(* PLC project conveyor, truST trust-runtime 0.24.54 *)
(* stored: creationDateTime 1786456263Z *)

TYPE XY : STRUCT
  X : lreal;
  Y : lreal;
END_STRUCT;
END_TYPE

FUNCTION RotateSquarePoints : XYPoints
VAR_IN_OUT
    Square : XYPoints;
END_VAR
VAR
   X : LREAL;
   Y : LREAL;
   I : INT;
END_VAR
FOR I := 0 TO 3 DO 
    X := Square[I].X;
    Y := Square[I].Y;
    Square[I] := RotateXY(
    X := X,
    Y := Y,
    THETA := 90.0
    );
END_FOR
RotateSquarePoints := Square;
END_FUNCTION

FUNCTION RotateSquarePoints : XYPoints
VAR_IN_OUT
    Square : XYPoints;
END_VAR
VAR
   X : LREAL;
   Y : LREAL;
   I : INT;
END_VAR
FOR I := 0 TO 3 DO 
    X := Square[I].X;
    Y := Square[I].Y;
    Square[I] := RotateXY(
    X := X,
    Y := Y,
    THETA := 90.0
    );
END_FOR
RotateSquarePoints := Square;
END_FUNCTION
END_FUNCTION

FUNCTION RotateXY : XY
VAR_INPUT
    X : LREAL;
    Y : LREAL;
    THETA : LREAL;
END_VAR
VAR
    Out : XY;
    SinM : LREAL;
    CosM : LREAL;
    THETA_RAD : LREAL;
END_VAR 
   
   THETA_RAD := REAL_TO_LREAL(
    RAD(
        LREAL_TO_REAL(THETA)
        )
    );  
   SinM := SIN(THETA_RAD);
   Cosm := COS(THETA_RAD);
   Out.X := X * CosM - Y * SinM;
   Out.Y := X * SinM + Y * CosM;
   RotateXY := Out;
END_FUNCTION

FUNCTION RotateXY : XY
VAR_INPUT
    X : LREAL;
    Y : LREAL;
    THETA : LREAL;
END_VAR
VAR
    Out : XY;
    SinM : LREAL;
    CosM : LREAL;
    THETA_RAD : LREAL;
END_VAR 
   
   THETA_RAD := REAL_TO_LREAL(
    RAD(
        LREAL_TO_REAL(THETA)
        )
    );  
   SinM := SIN(THETA_RAD);
   Cosm := COS(THETA_RAD);
   Out.X := X * CosM - Y * SinM;
   Out.Y := X * SinM + Y * CosM;
   RotateXY := Out;
END_FUNCTION
END_FUNCTION

FUNCTION SquarePoints : XYPoints
VAR_OUTPUT
    //Square : Array[0..1] of LREAL;//XYPoints;
END_VAR
VAR_INPUT
    Length : LREAL := 5.0;
    
END_VAR
VAR
   Zero : LREAL := 0.0;
   Square : XYPoints;
END_VAR

    Square[0].X := Zero;
    Square[0].Y := Length;
    Square[1].X := Length;
    Square[1].Y := Length;    
    Square[2].X := Length;
    Square[2].Y := Zero;
    Square[3].X := Zero;
    Square[3].Y := Zero; 
    SquarePoints := Square;
END_FUNCTION

FUNCTION SquarePoints : XYPoints
VAR_OUTPUT
    //Square : Array[0..1] of LREAL;//XYPoints;
END_VAR
VAR_INPUT
    Length : LREAL := 5.0;
    
END_VAR
VAR
   Zero : LREAL := 0.0;
   Square : XYPoints;
END_VAR

    Square[0].X := Zero;
    Square[0].Y := Length;
    Square[1].X := Length;
    Square[1].Y := Length;    
    Square[2].X := Length;
    Square[2].Y := Zero;
    Square[3].X := Zero;
    Square[3].Y := Zero; 
    SquarePoints := Square;
END_FUNCTION
END_FUNCTION

PROGRAM MainProgram
VAR
    e_stop         : BOOL;   (* %IX0.0 — write TRUE to stop the line *)
    running        : BOOL;   (* %QX2.0 *)
    conveyor_speed : INT;    (* %QW0   *)
    part_count     : INT;    (* %MW0   *)
    out : XYPoints;
    Length : LREAL := 5.0;
END_VAR

out := SquarePoints();//Length := Length);//, Square => out); 
RotateSquarePoints(Square := out);
running := NOT e_stop;
IF running THEN
    IF conveyor_speed < 100 THEN
        conveyor_speed := conveyor_speed + 5;
    ELSE
        part_count := part_count + 1;
        conveyor_speed := 0;
    END_IF;
ELSE
    conveyor_speed := 0;
END_IF;
END_PROGRAM

PROGRAM MainProgram
VAR
    e_stop         : BOOL;   (* %IX0.0 — write TRUE to stop the line *)
    running        : BOOL;   (* %QX2.0 *)
    conveyor_speed : INT;    (* %QW0   *)
    part_count     : INT;    (* %MW0   *)
    out : XYPoints;
    Length : LREAL := 5.0;
END_VAR

out := SquarePoints();//Length := Length);//, Square => out); 
RotateSquarePoints(Square := out);
running := NOT e_stop;
IF running THEN
    IF conveyor_speed < 100 THEN
        conveyor_speed := conveyor_speed + 5;
    ELSE
        part_count := part_count + 1;
        conveyor_speed := 0;
    END_IF;
ELSE
    conveyor_speed := 0;
END_IF;
END_PROGRAM
END_PROGRAM

FUNCTION RotateSquarePoints : XYPoints
VAR_IN_OUT
    Square : XYPoints;
END_VAR
VAR
   X : LREAL;
   Y : LREAL;
   I : INT;
END_VAR
FOR I := 0 TO 3 DO 
    X := Square[I].X;
    Y := Square[I].Y;
    Square[I] := RotateXY(
    X := X,
    Y := Y,
    THETA := 90.0
    );
END_FOR
RotateSquarePoints := Square;
END_FUNCTION

                  FUNCTION RotateSquarePoints : XYPoints
VAR_IN_OUT
    Square : XYPoints;
END_VAR
VAR
   X : LREAL;
   Y : LREAL;
   I : INT;
END_VAR
FOR I := 0 TO 3 DO 
    X := Square[I].X;
    Y := Square[I].Y;
    Square[I] := RotateXY(
    X := X,
    Y := Y,
    THETA := 90.0
    );
END_FOR
RotateSquarePoints := Square;
END_FUNCTION

                
END_FUNCTION

FUNCTION RotateXY : XY
VAR_INPUT
    X : LREAL;
    Y : LREAL;
    THETA : LREAL;
END_VAR
VAR
    Out : XY;
    SinM : LREAL;
    CosM : LREAL;
    THETA_RAD : LREAL;
END_VAR 
   
   THETA_RAD := REAL_TO_LREAL(
    RAD(
        LREAL_TO_REAL(THETA)
        )
    );  
   SinM := SIN(THETA_RAD);
   Cosm := COS(THETA_RAD);
   Out.X := X * CosM - Y * SinM;
   Out.Y := X * SinM + Y * CosM;
   RotateXY := Out;
END_FUNCTION

                  FUNCTION RotateXY : XY
VAR_INPUT
    X : LREAL;
    Y : LREAL;
    THETA : LREAL;
END_VAR
VAR
    Out : XY;
    SinM : LREAL;
    CosM : LREAL;
    THETA_RAD : LREAL;
END_VAR 
   
   THETA_RAD := REAL_TO_LREAL(
    RAD(
        LREAL_TO_REAL(THETA)
        )
    );  
   SinM := SIN(THETA_RAD);
   Cosm := COS(THETA_RAD);
   Out.X := X * CosM - Y * SinM;
   Out.Y := X * SinM + Y * CosM;
   RotateXY := Out;
END_FUNCTION

                
END_FUNCTION

FUNCTION SquarePoints : XYPoints
VAR_OUTPUT
    //Square : Array[0..1] of LREAL;//XYPoints;
END_VAR
VAR_INPUT
    Length : LREAL := 5.0;
    
END_VAR
VAR
   Zero : LREAL := 0.0;
   Square : XYPoints;
END_VAR

    Square[0].X := Zero;
    Square[0].Y := Length;
    Square[1].X := Length;
    Square[1].Y := Length;    
    Square[2].X := Length;
    Square[2].Y := Zero;
    Square[3].X := Zero;
    Square[3].Y := Zero; 
    SquarePoints := Square;
END_FUNCTION

                  FUNCTION SquarePoints : XYPoints
VAR_OUTPUT
    //Square : Array[0..1] of LREAL;//XYPoints;
END_VAR
VAR_INPUT
    Length : LREAL := 5.0;
    
END_VAR
VAR
   Zero : LREAL := 0.0;
   Square : XYPoints;
END_VAR

    Square[0].X := Zero;
    Square[0].Y := Length;
    Square[1].X := Length;
    Square[1].Y := Length;    
    Square[2].X := Length;
    Square[2].Y := Zero;
    Square[3].X := Zero;
    Square[3].Y := Zero; 
    SquarePoints := Square;
END_FUNCTION

                
END_FUNCTION

PROGRAM MainProgram
VAR
    e_stop         : BOOL;   (* %IX0.0 — write TRUE to stop the line *)
    running        : BOOL;   (* %QX2.0 *)
    conveyor_speed : INT;    (* %QW0   *)
    part_count     : INT;    (* %MW0   *)
    out : XYPoints;
    Length : LREAL := 5.0;
END_VAR

out := SquarePoints();//Length := Length);//, Square => out); 
RotateSquarePoints(Square := out);
running := NOT e_stop;
IF running THEN
    IF conveyor_speed < 100 THEN
        conveyor_speed := conveyor_speed + 5;
    ELSE
        part_count := part_count + 1;
        conveyor_speed := 0;
    END_IF;
ELSE
    conveyor_speed := 0;
END_IF;
END_PROGRAM

                  
PROGRAM MainProgram
VAR
    e_stop         : BOOL;   (* %IX0.0 — write TRUE to stop the line *)
    running        : BOOL;   (* %QX2.0 *)
    conveyor_speed : INT;    (* %QW0   *)
    part_count     : INT;    (* %MW0   *)
    out : XYPoints;
    Length : LREAL := 5.0;
END_VAR

out := SquarePoints();//Length := Length);//, Square => out); 
RotateSquarePoints(Square := out);
running := NOT e_stop;
IF running THEN
    IF conveyor_speed < 100 THEN
        conveyor_speed := conveyor_speed + 5;
    ELSE
        part_count := part_count + 1;
        conveyor_speed := 0;
    END_IF;
ELSE
    conveyor_speed := 0;
END_IF;
END_PROGRAM


                
END_PROGRAM

CONFIGURATION ConveyorCell
END_CONFIGURATION
